ABB RAPID module: MainModule.mod

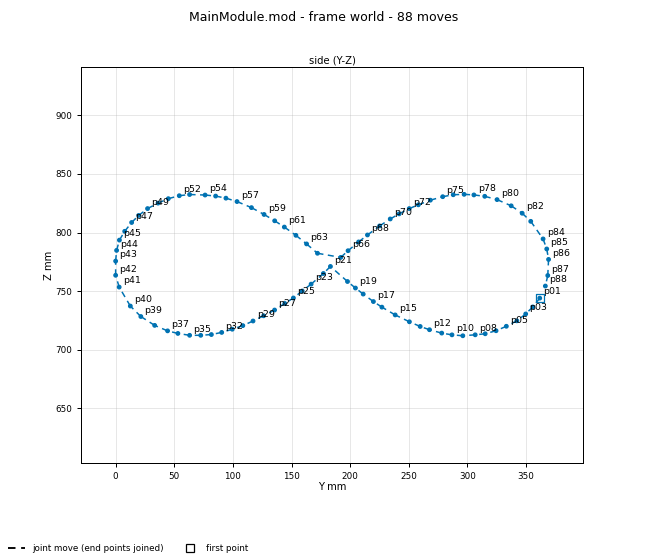
[picture p0: tool path of MainModule.mod in frame world, 88 of 88 moves have a stored position in this frame; points joined in program order, loops and branches not executed]
MODULE MainModule
	CONST robtarget p01 := [ [500.0, 361.64814814814815, 744.0909090909091], [0.707106781, 0, 0.707106781, 0], [0, 0, 0, 0], [ 9E9, 9E9, 9E9, 9E9, 9E9, 9E9] ];
	CONST robtarget p02 := [ [500.0, 355.64814814814815, 736.5909090909091], [0.707106781, 0, 0.707106781, 0], [0, 0, 0, 0], [ 9E9, 9E9, 9E9, 9E9, 9E9, 9E9] ];
	CONST robtarget p03 := [ [500.0, 349.64814814814815, 730.5909090909091], [0.707106781, 0, 0.707106781, 0], [0, 0, 0, 0], [ 9E9, 9E9, 9E9, 9E9, 9E9, 9E9] ];
	CONST robtarget p04 := [ [500.0, 342.08363201911584, 724.7360703812317], [0.707106781, 0, 0.707106781, 0], [0, 0, 0, 0], [ 9E9, 9E9, 9E9, 9E9, 9E9, 9E9] ];
	CONST robtarget p05 := [ [500.0, 333.14814814814815, 720.0909090909091], [0.707106781, 0, 0.707106781, 0], [0, 0, 0, 0], [ 9E9, 9E9, 9E9, 9E9, 9E9, 9E9] ];
	CONST robtarget p06 := [ [500.0, 324.3722860791827, 716.2805642633228], [0.707106781, 0, 0.707106781, 0], [0, 0, 0, 0], [ 9E9, 9E9, 9E9, 9E9, 9E9, 9E9] ];
	CONST robtarget p07 := [ [500.0, 315.1111111111111, 713.7020202020202], [0.707106781, 0, 0.707106781, 0], [0, 0, 0, 0], [ 9E9, 9E9, 9E9, 9E9, 9E9, 9E9] ];
	CONST robtarget p08 := [ [500.0, 306.5940940940941, 712.813882063882], [0.707106781, 0, 0.707106781, 0], [0, 0, 0, 0], [ 9E9, 9E9, 9E9, 9E9, 9E9, 9E9] ];
	CONST robtarget p09 := [ [500.0, 296.0345117845118, 712.0], [0.707106781, 0, 0.707106781, 0], [0, 0, 0, 0], [ 9E9, 9E9, 9E9, 9E9, 9E9, 9E9] ];
	CONST robtarget p10 := [ [500.0, 286.78877314814815, 712.7784090909091], [0.707106781, 0, 0.707106781, 0], [0, 0, 0, 0], [ 9E9, 9E9, 9E9, 9E9, 9E9, 9E9] ];
	CONST robtarget p11 := [ [500.0, 278.0619412515964, 714.2719435736677], [0.707106781, 0, 0.707106781, 0], [0, 0, 0, 0], [ 9E9, 9E9, 9E9, 9E9, 9E9, 9E9] ];
	CONST robtarget p12 := [ [500.0, 267.6187363834423, 717.1497326203208], [0.707106781, 0, 0.707106781, 0], [0, 0, 0, 0], [ 9E9, 9E9, 9E9, 9E9, 9E9, 9E9] ];
	CONST robtarget p13 := [ [500.0, 259.6800630417652, 719.931334622824], [0.707106781, 0, 0.707106781, 0], [0, 0, 0, 0], [ 9E9, 9E9, 9E9, 9E9, 9E9, 9E9] ];
	CONST robtarget p14 := [ [500.0, 250.48148148148147, 723.9242424242425], [0.707106781, 0, 0.707106781, 0], [0, 0, 0, 0], [ 9E9, 9E9, 9E9, 9E9, 9E9, 9E9] ];
	CONST robtarget p15 := [ [500.0, 238.36243386243382, 729.7694805194806], [0.707106781, 0, 0.707106781, 0], [0, 0, 0, 0], [ 9E9, 9E9, 9E9, 9E9, 9E9, 9E9] ];
	CONST robtarget p16 := [ [500.0, 227.04100529100526, 736.4123376623377], [0.707106781, 0, 0.707106781, 0], [0, 0, 0, 0], [ 9E9, 9E9, 9E9, 9E9, 9E9, 9E9] ];
	CONST robtarget p17 := [ [500.0, 219.79100529100526, 741.1623376623377], [0.707106781, 0, 0.707106781, 0], [0, 0, 0, 0], [ 9E9, 9E9, 9E9, 9E9, 9E9, 9E9] ];
	CONST robtarget p18 := [ [500.0, 211.09000861326444, 747.5443974630022], [0.707106781, 0, 0.707106781, 0], [0, 0, 0, 0], [ 9E9, 9E9, 9E9, 9E9, 9E9, 9E9] ];
	CONST robtarget p19 := [ [500.0, 204.4621016365203, 752.7071881606765], [0.707106781, 0, 0.707106781, 0], [0, 0, 0, 0], [ 9E9, 9E9, 9E9, 9E9, 9E9, 9E9] ];
	CONST robtarget p20 := [ [500.0, 197.6981481481481, 758.2659090909091], [0.707106781, 0, 0.707106781, 0], [0, 0, 0, 0], [ 9E9, 9E9, 9E9, 9E9, 9E9, 9E9] ];
	CONST robtarget p21 := [ [500.0, 183.14814814814815, 771.0909090909091], [0.707106781, 0, 0.707106781, 0], [0, 0, 0, 0], [ 9E9, 9E9, 9E9, 9E9, 9E9, 9E9] ];
	CONST robtarget p22 := [ [500.0, 177.14814814814815, 765.0909090909091], [0.707106781, 0, 0.707106781, 0], [0, 0, 0, 0], [ 9E9, 9E9, 9E9, 9E9, 9E9, 9E9] ];
	CONST robtarget p23 := [ [500.0, 166.67939814814815, 756.0127840909091], [0.707106781, 0, 0.707106781, 0], [0, 0, 0, 0], [ 9E9, 9E9, 9E9, 9E9, 9E9, 9E9] ];
	CONST robtarget p24 := [ [500.0, 159.11689814814815, 750.1690340909091], [0.707106781, 0, 0.707106781, 0], [0, 0, 0, 0], [ 9E9, 9E9, 9E9, 9E9, 9E9, 9E9] ];
	CONST robtarget p25 := [ [500.0, 151.5692007797271, 744.233014354067], [0.707106781, 0, 0.707106781, 0], [0, 0, 0, 0], [ 9E9, 9E9, 9E9, 9E9, 9E9, 9E9] ];
	CONST robtarget p26 := [ [500.0, 144.1960204885737, 739.527079303675], [0.707106781, 0, 0.707106781, 0], [0, 0, 0, 0], [ 9E9, 9E9, 9E9, 9E9, 9E9, 9E9] ];
	CONST robtarget p27 := [ [500.0, 135.52314814814815, 733.949604743083], [0.707106781, 0, 0.707106781, 0], [0, 0, 0, 0], [ 9E9, 9E9, 9E9, 9E9, 9E9, 9E9] ];
	CONST robtarget p28 := [ [500.0, 126.19706119162642, 729.0256916996047], [0.707106781, 0, 0.707106781, 0], [0, 0, 0, 0], [ 9E9, 9E9, 9E9, 9E9, 9E9, 9E9] ];
	CONST robtarget p29 := [ [500.0, 117.14814814814814, 724.5909090909091], [0.707106781, 0, 0.707106781, 0], [0, 0, 0, 0], [ 9E9, 9E9, 9E9, 9E9, 9E9, 9E9] ];
	CONST robtarget p30 := [ [500.0, 108.45151893466497, 720.64708886619], [0.707106781, 0, 0.707106781, 0], [0, 0, 0, 0], [ 9E9, 9E9, 9E9, 9E9, 9E9, 9E9] ];
	CONST robtarget p31 := [ [500.0, 99.45496632996633, 717.5681818181818], [0.707106781, 0, 0.707106781, 0], [0, 0, 0, 0], [ 9E9, 9E9, 9E9, 9E9, 9E9, 9E9] ];
	CONST robtarget p32 := [ [500.0, 90.43386243386242, 714.8587662337662], [0.707106781, 0, 0.707106781, 0], [0, 0, 0, 0], [ 9E9, 9E9, 9E9, 9E9, 9E9, 9E9] ];
	CONST robtarget p33 := [ [500.0, 81.63516113516111, 713.038961038961], [0.707106781, 0, 0.707106781, 0], [0, 0, 0, 0], [ 9E9, 9E9, 9E9, 9E9, 9E9, 9E9] ];
	CONST robtarget p34 := [ [500.0, 72.56726579520698, 712.3923796791444], [0.707106781, 0, 0.707106781, 0], [0, 0, 0, 0], [ 9E9, 9E9, 9E9, 9E9, 9E9, 9E9] ];
	CONST robtarget p35 := [ [500.0, 63.079966329966325, 712.3863636363636], [0.707106781, 0, 0.707106781, 0], [0, 0, 0, 0], [ 9E9, 9E9, 9E9, 9E9, 9E9, 9E9] ];
	CONST robtarget p36 := [ [500.0, 53.08780332056192, 713.987460815047], [0.707106781, 0, 0.707106781, 0], [0, 0, 0, 0], [ 9E9, 9E9, 9E9, 9E9, 9E9, 9E9] ];
	CONST robtarget p37 := [ [500.0, 44.29520697167756, 716.1791443850268], [0.707106781, 0, 0.707106781, 0], [0, 0, 0, 0], [ 9E9, 9E9, 9E9, 9E9, 9E9, 9E9] ];
	CONST robtarget p38 := [ [500.0, 33.281481481481464, 720.8575757575758], [0.707106781, 0, 0.707106781, 0], [0, 0, 0, 0], [ 9E9, 9E9, 9E9, 9E9, 9E9, 9E9] ];
	CONST robtarget p39 := [ [500.0, 21.48905723905723, 728.4090909090909], [0.707106781, 0, 0.707106781, 0], [0, 0, 0, 0], [ 9E9, 9E9, 9E9, 9E9, 9E9, 9E9] ];
	CONST robtarget p40 := [ [500.0, 12.523148148148138, 737.3409090909091], [0.707106781, 0, 0.707106781, 0], [0, 0, 0, 0], [ 9E9, 9E9, 9E9, 9E9, 9E9, 9E9] ];
	CONST robtarget p41 := [ [500.0, 3.0195767195767047, 753.498051948052], [0.707106781, 0, 0.707106781, 0], [0, 0, 0, 0], [ 9E9, 9E9, 9E9, 9E9, 9E9, 9E9] ];
	CONST robtarget p42 := [ [500.0, 1.9336549319050237e-31, 763.5723905723905], [0.707106781, 0, 0.707106781, 0], [0, 0, 0, 0], [ 9E9, 9E9, 9E9, 9E9, 9E9, 9E9] ];
	CONST robtarget p43 := [ [500.0, 0.006971677559903355, 775.6791443850268], [0.707106781, 0, 0.707106781, 0], [0, 0, 0, 0], [ 9E9, 9E9, 9E9, 9E9, 9E9, 9E9] ];
	CONST robtarget p44 := [ [500.0, 0.8270955165691731, 784.7961722488038], [0.707106781, 0, 0.707106781, 0], [0, 0, 0, 0], [ 9E9, 9E9, 9E9, 9E9, 9E9, 9E9] ];
	CONST robtarget p45 := [ [500.0, 3.226273148148138, 793.5596590909091], [0.707106781, 0, 0.707106781, 0], [0, 0, 0, 0], [ 9E9, 9E9, 9E9, 9E9, 9E9, 9E9] ];
	CONST robtarget p46 := [ [500.0, 7.726273148148138, 801.0596590909091], [0.707106781, 0, 0.707106781, 0], [0, 0, 0, 0], [ 9E9, 9E9, 9E9, 9E9, 9E9, 9E9] ];
	CONST robtarget p47 := [ [500.0, 13.648148148148138, 808.5909090909091], [0.707106781, 0, 0.707106781, 0], [0, 0, 0, 0], [ 9E9, 9E9, 9E9, 9E9, 9E9, 9E9] ];
	CONST robtarget p48 := [ [500.0, 19.648148148148138, 814.5909090909091], [0.707106781, 0, 0.707106781, 0], [0, 0, 0, 0], [ 9E9, 9E9, 9E9, 9E9, 9E9, 9E9] ];
	CONST robtarget p49 := [ [500.0, 27.212664277180394, 820.4457478005866], [0.707106781, 0, 0.707106781, 0], [0, 0, 0, 0], [ 9E9, 9E9, 9E9, 9E9, 9E9, 9E9] ];
	CONST robtarget p50 := [ [500.0, 36.14814814814814, 825.0909090909091], [0.707106781, 0, 0.707106781, 0], [0, 0, 0, 0], [ 9E9, 9E9, 9E9, 9E9, 9E9, 9E9] ];
	CONST robtarget p51 := [ [500.0, 44.92401021711366, 828.9012539184953], [0.707106781, 0, 0.707106781, 0], [0, 0, 0, 0], [ 9E9, 9E9, 9E9, 9E9, 9E9, 9E9] ];
	CONST robtarget p52 := [ [500.0, 54.25790424570913, 831.420177383592], [0.707106781, 0, 0.707106781, 0], [0, 0, 0, 0], [ 9E9, 9E9, 9E9, 9E9, 9E9, 9E9] ];
	CONST robtarget p53 := [ [500.0, 63.048148148148144, 832.4309090909092], [0.707106781, 0, 0.707106781, 0], [0, 0, 0, 0], [ 9E9, 9E9, 9E9, 9E9, 9E9, 9E9] ];
	CONST robtarget p54 := [ [500.0, 76.26178451178451, 832.0], [0.707106781, 0, 0.707106781, 0], [0, 0, 0, 0], [ 9E9, 9E9, 9E9, 9E9, 9E9, 9E9] ];
	CONST robtarget p55 := [ [500.0, 85.26679221594473, 831.1163328197226], [0.707106781, 0, 0.707106781, 0], [0, 0, 0, 0], [ 9E9, 9E9, 9E9, 9E9, 9E9, 9E9] ];
	CONST robtarget p56 := [ [500.0, 94.04237891737891, 829.3312937062936], [0.707106781, 0, 0.707106781, 0], [0, 0, 0, 0], [ 9E9, 9E9, 9E9, 9E9, 9E9, 9E9] ];
	CONST robtarget p57 := [ [500.0, 103.48510466988726, 826.4278656126482], [0.707106781, 0, 0.707106781, 0], [0, 0, 0, 0], [ 9E9, 9E9, 9E9, 9E9, 9E9, 9E9] ];
	CONST robtarget p58 := [ [500.0, 115.81481481481482, 821.2575757575758], [0.707106781, 0, 0.707106781, 0], [0, 0, 0, 0], [ 9E9, 9E9, 9E9, 9E9, 9E9, 9E9] ];
	CONST robtarget p59 := [ [500.0, 126.56675279931092, 815.4281183932346], [0.707106781, 0, 0.707106781, 0], [0, 0, 0, 0], [ 9E9, 9E9, 9E9, 9E9, 9E9, 9E9] ];
	CONST robtarget p60 := [ [500.0, 135.62542087542084, 810.0227272727273], [0.707106781, 0, 0.707106781, 0], [0, 0, 0, 0], [ 9E9, 9E9, 9E9, 9E9, 9E9, 9E9] ];
	CONST robtarget p61 := [ [500.0, 143.84814814814814, 804.6909090909091], [0.707106781, 0, 0.707106781, 0], [0, 0, 0, 0], [ 9E9, 9E9, 9E9, 9E9, 9E9, 9E9] ];
	CONST robtarget p62 := [ [500.0, 153.70628768303186, 797.6374207188161], [0.707106781, 0, 0.707106781, 0], [0, 0, 0, 0], [ 9E9, 9E9, 9E9, 9E9, 9E9, 9E9] ];
	CONST robtarget p63 := [ [500.0, 162.7958754208754, 790.3181818181818], [0.707106781, 0, 0.707106781, 0], [0, 0, 0, 0], [ 9E9, 9E9, 9E9, 9E9, 9E9, 9E9] ];
	CONST robtarget p64 := [ [500.0, 172.11243386243387, 782.3409090909091], [0.707106781, 0, 0.707106781, 0], [0, 0, 0, 0], [ 9E9, 9E9, 9E9, 9E9, 9E9, 9E9] ];
	CONST robtarget p65 := [ [500.0, 191.92234169653523, 778.816715542522], [0.707106781, 0, 0.707106781, 0], [0, 0, 0, 0], [ 9E9, 9E9, 9E9, 9E9, 9E9, 9E9] ];
	CONST robtarget p66 := [ [500.0, 198.17939814814815, 784.5127840909091], [0.707106781, 0, 0.707106781, 0], [0, 0, 0, 0], [ 9E9, 9E9, 9E9, 9E9, 9E9, 9E9] ];
	CONST robtarget p67 := [ [500.0, 207.17939814814815, 792.0127840909091], [0.707106781, 0, 0.707106781, 0], [0, 0, 0, 0], [ 9E9, 9E9, 9E9, 9E9, 9E9, 9E9] ];
	CONST robtarget p68 := [ [500.0, 214.7270955165692, 797.9488038277511], [0.707106781, 0, 0.707106781, 0], [0, 0, 0, 0], [ 9E9, 9E9, 9E9, 9E9, 9E9, 9E9] ];
	CONST robtarget p69 := [ [500.0, 225.1002758077226, 805.6547388781431], [0.707106781, 0, 0.707106781, 0], [0, 0, 0, 0], [ 9E9, 9E9, 9E9, 9E9, 9E9, 9E9] ];
	CONST robtarget p70 := [ [500.0, 234.14814814814815, 811.5909090909091], [0.707106781, 0, 0.707106781, 0], [0, 0, 0, 0], [ 9E9, 9E9, 9E9, 9E9, 9E9, 9E9] ];
	CONST robtarget p71 := [ [500.0, 241.7126642771804, 815.9457478005866], [0.707106781, 0, 0.707106781, 0], [0, 0, 0, 0], [ 9E9, 9E9, 9E9, 9E9, 9E9, 9E9] ];
	CONST robtarget p72 := [ [500.0, 250.37848522679985, 820.4392236976507], [0.707106781, 0, 0.707106781, 0], [0, 0, 0, 0], [ 9E9, 9E9, 9E9, 9E9, 9E9, 9E9] ];
	CONST robtarget p73 := [ [500.0, 258.0992351046699, 823.6561264822135], [0.707106781, 0, 0.707106781, 0], [0, 0, 0, 0], [ 9E9, 9E9, 9E9, 9E9, 9E9, 9E9] ];
	CONST robtarget p74 := [ [500.0, 268.34132996632997, 827.6136363636364], [0.707106781, 0, 0.707106781, 0], [0, 0, 0, 0], [ 9E9, 9E9, 9E9, 9E9, 9E9, 9E9] ];
	CONST robtarget p75 := [ [500.0, 278.89205058717255, 830.5787139689579], [0.707106781, 0, 0.707106781, 0], [0, 0, 0, 0], [ 9E9, 9E9, 9E9, 9E9, 9E9, 9E9] ];
	CONST robtarget p76 := [ [500.0, 287.8520955165692, 832.2356459330143], [0.707106781, 0, 0.707106781, 0], [0, 0, 0, 0], [ 9E9, 9E9, 9E9, 9E9, 9E9, 9E9] ];
	CONST robtarget p77 := [ [500.0, 297.14814814814815, 832.5909090909091], [0.707106781, 0, 0.707106781, 0], [0, 0, 0, 0], [ 9E9, 9E9, 9E9, 9E9, 9E9, 9E9] ];
	CONST robtarget p78 := [ [500.0, 305.4789173789174, 832.0832167832168], [0.707106781, 0, 0.707106781, 0], [0, 0, 0, 0], [ 9E9, 9E9, 9E9, 9E9, 9E9, 9E9] ];
	CONST robtarget p79 := [ [500.0, 314.7343550446999, 830.9098746081505], [0.707106781, 0, 0.707106781, 0], [0, 0, 0, 0], [ 9E9, 9E9, 9E9, 9E9, 9E9, 9E9] ];
	CONST robtarget p80 := [ [500.0, 325.2281481481482, 828.0909090909091], [0.707106781, 0, 0.707106781, 0], [0, 0, 0, 0], [ 9E9, 9E9, 9E9, 9E9, 9E9, 9E9] ];
	CONST robtarget p81 := [ [500.0, 337.27314814814815, 822.8068181818181], [0.707106781, 0, 0.707106781, 0], [0, 0, 0, 0], [ 9E9, 9E9, 9E9, 9E9, 9E9, 9E9] ];
	CONST robtarget p82 := [ [500.0, 346.64814814814815, 816.4659090909091], [0.707106781, 0, 0.707106781, 0], [0, 0, 0, 0], [ 9E9, 9E9, 9E9, 9E9, 9E9, 9E9] ];
	CONST robtarget p83 := [ [500.0, 353.95249597423515, 809.5691699604743], [0.707106781, 0, 0.707106781, 0], [0, 0, 0, 0], [ 9E9, 9E9, 9E9, 9E9, 9E9, 9E9] ];
	CONST robtarget p84 := [ [500.0, 364.4690436705363, 794.5759837177748], [0.707106781, 0, 0.707106781, 0], [0, 0, 0, 0], [ 9E9, 9E9, 9E9, 9E9, 9E9, 9E9] ];
	CONST robtarget p85 := [ [500.0, 367.5918981481481, 786.0159090909091], [0.707106781, 0, 0.707106781, 0], [0, 0, 0, 0], [ 9E9, 9E9, 9E9, 9E9, 9E9, 9E9] ];
	CONST robtarget p86 := [ [500.0, 369.14814814814815, 777.0909090909091], [0.707106781, 0, 0.707106781, 0], [0, 0, 0, 0], [ 9E9, 9E9, 9E9, 9E9, 9E9, 9E9] ];
	CONST robtarget p87 := [ [500.0, 368.4692007797271, 763.3856459330143], [0.707106781, 0, 0.707106781, 0], [0, 0, 0, 0], [ 9E9, 9E9, 9E9, 9E9, 9E9, 9E9] ];
	CONST robtarget p88 := [ [500.0, 366.4007797270955, 754.4014354066985], [0.707106781, 0, 0.707106781, 0], [0, 0, 0, 0], [ 9E9, 9E9, 9E9, 9E9, 9E9, 9E9] ];
	PROC main()
		MoveJ p01, v200, z20, tool0;
		MoveJ p02, v200, z20, tool0;
		MoveJ p03, v200, z20, tool0;
		MoveJ p04, v200, z20, tool0;
		MoveJ p05, v200, z20, tool0;
		MoveJ p06, v200, z20, tool0;
		MoveJ p07, v200, z20, tool0;
		MoveJ p08, v200, z20, tool0;
		MoveJ p09, v200, z20, tool0;
		MoveJ p10, v200, z20, tool0;
		MoveJ p11, v200, z20, tool0;
		MoveJ p12, v200, z20, tool0;
		MoveJ p13, v200, z20, tool0;
		MoveJ p14, v200, z20, tool0;
		MoveJ p15, v200, z20, tool0;
		MoveJ p16, v200, z20, tool0;
		MoveJ p17, v200, z20, tool0;
		MoveJ p18, v200, z20, tool0;
		MoveJ p19, v200, z20, tool0;
		MoveJ p20, v200, z20, tool0;
		MoveJ p21, v200, z20, tool0;
		MoveJ p22, v200, z20, tool0;
		MoveJ p23, v200, z20, tool0;
		MoveJ p24, v200, z20, tool0;
		MoveJ p25, v200, z20, tool0;
		MoveJ p26, v200, z20, tool0;
		MoveJ p27, v200, z20, tool0;
		MoveJ p28, v200, z20, tool0;
		MoveJ p29, v200, z20, tool0;
		MoveJ p30, v200, z20, tool0;
		MoveJ p31, v200, z20, tool0;
		MoveJ p32, v200, z20, tool0;
		MoveJ p33, v200, z20, tool0;
		MoveJ p34, v200, z20, tool0;
		MoveJ p35, v200, z20, tool0;
		MoveJ p36, v200, z20, tool0;
		MoveJ p37, v200, z20, tool0;
		MoveJ p38, v200, z20, tool0;
		MoveJ p39, v200, z20, tool0;
		MoveJ p40, v200, z20, tool0;
		MoveJ p41, v200, z20, tool0;
		MoveJ p42, v200, z20, tool0;
		MoveJ p43, v200, z20, tool0;
		MoveJ p44, v200, z20, tool0;
		MoveJ p45, v200, z20, tool0;
		MoveJ p46, v200, z20, tool0;
		MoveJ p47, v200, z20, tool0;
		MoveJ p48, v200, z20, tool0;
		MoveJ p49, v200, z20, tool0;
		MoveJ p50, v200, z20, tool0;
		MoveJ p51, v200, z20, tool0;
		MoveJ p52, v200, z20, tool0;
		MoveJ p53, v200, z20, tool0;
		MoveJ p54, v200, z20, tool0;
		MoveJ p55, v200, z20, tool0;
		MoveJ p56, v200, z20, tool0;
		MoveJ p57, v200, z20, tool0;
		MoveJ p58, v200, z20, tool0;
		MoveJ p59, v200, z20, tool0;
		MoveJ p60, v200, z20, tool0;
		MoveJ p61, v200, z20, tool0;
		MoveJ p62, v200, z20, tool0;
		MoveJ p63, v200, z20, tool0;
		MoveJ p64, v200, z20, tool0;
		MoveJ p65, v200, z20, tool0;
		MoveJ p66, v200, z20, tool0;
		MoveJ p67, v200, z20, tool0;
		MoveJ p68, v200, z20, tool0;
		MoveJ p69, v200, z20, tool0;
		MoveJ p70, v200, z20, tool0;
		MoveJ p71, v200, z20, tool0;
		MoveJ p72, v200, z20, tool0;
		MoveJ p73, v200, z20, tool0;
		MoveJ p74, v200, z20, tool0;
		MoveJ p75, v200, z20, tool0;
		MoveJ p76, v200, z20, tool0;
		MoveJ p77, v200, z20, tool0;
		MoveJ p78, v200, z20, tool0;
		MoveJ p79, v200, z20, tool0;
		MoveJ p80, v200, z20, tool0;
		MoveJ p81, v200, z20, tool0;
		MoveJ p82, v200, z20, tool0;
		MoveJ p83, v200, z20, tool0;
		MoveJ p84, v200, z20, tool0;
		MoveJ p85, v200, z20, tool0;
		MoveJ p86, v200, z20, tool0;
		MoveJ p87, v200, z20, tool0;
		MoveJ p88, v200, z20, tool0;
	ENDPROC
ENDMODULE
